FUNCTION_BLOCK TickGen
  (* Standard: 61499-2 *)
  (* Version 0.1, 2017-00-25, hpea485, UOA *)
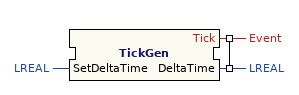
  EVENT_OUTPUT
    Tick WITH DeltaTime;
  END_EVENT
  VAR_INPUT
    SetDeltaTime : LREAL;
  END_VAR
  VAR_OUTPUT
    DeltaTime : LREAL;
  END_VAR
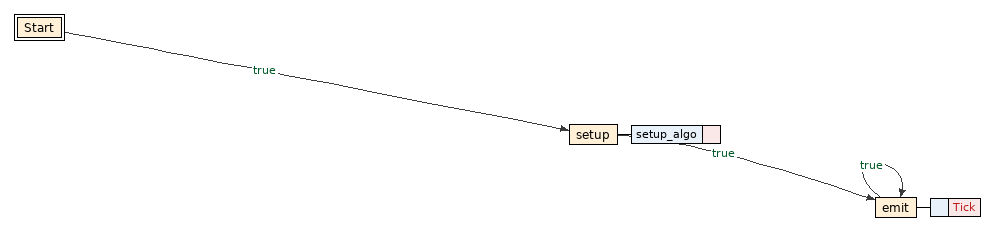
  EC_STATES
    Start;
    setup : setup_algo;
    emit : -> Tick;
  END_STATES
  EC_TRANSITIONS
    Start TO setup := true;
    setup TO emit := true;
    emit TO emit := true;
  END_TRANSITIONS
  ALGORITHM setup_algo IN C:
me->DeltaTime = me->SetDeltaTime;
  END_ALGORITHM
END_FUNCTION_BLOCK
